/// container for all communication data types that are used by the unit
TYPE QualityInspectionComRef :
STRUCT
  Publish : REFERENCE TO QualityInspectionComPublish; 
  Subscribe : REFERENCE TO QualityInspectionComSubscribe; 
END_STRUCT
END_TYPE

(* stored: Version 1.1.0.1
   DUT QualityInspectionComRef: Id {7fc5393d-3693-429e-a9f3-dd5517ac3e08} *)
